// LS Electric XG5000 project: 121대대(4-11-23)
// PLC NewPLC
// module base 0 slot 0: 16점 예약 할당:XG-IN16
// module base 0 slot 1: Cnet:XGL-CH2A/B (Cnet 통신 모듈(RS-232C, RS-422/485))
// module base 0 slot 2: 아날로그입력 모듈:XGF-AC8A (A/D 전류 입력형 8채널)
// module base 0 slot 3: 입력 모듈:XGI-D24A/B (DC 24V 입력, 32점 (전류소스 싱크공용/ 전류소스 입력))
// module base 0 slot 4: 출력 모듈:XGQ-TR4A/B (트랜지스터 출력, 32점 (0.1A용, 싱크출력/소스출력))
// module base 0 slot 5: 고속카운터 모듈:XGF-HO2A (고속카운터 펄스(OC) 입력형, 2채널)

PROGRAM Sequence_Program (task: 스캔 프로그램)

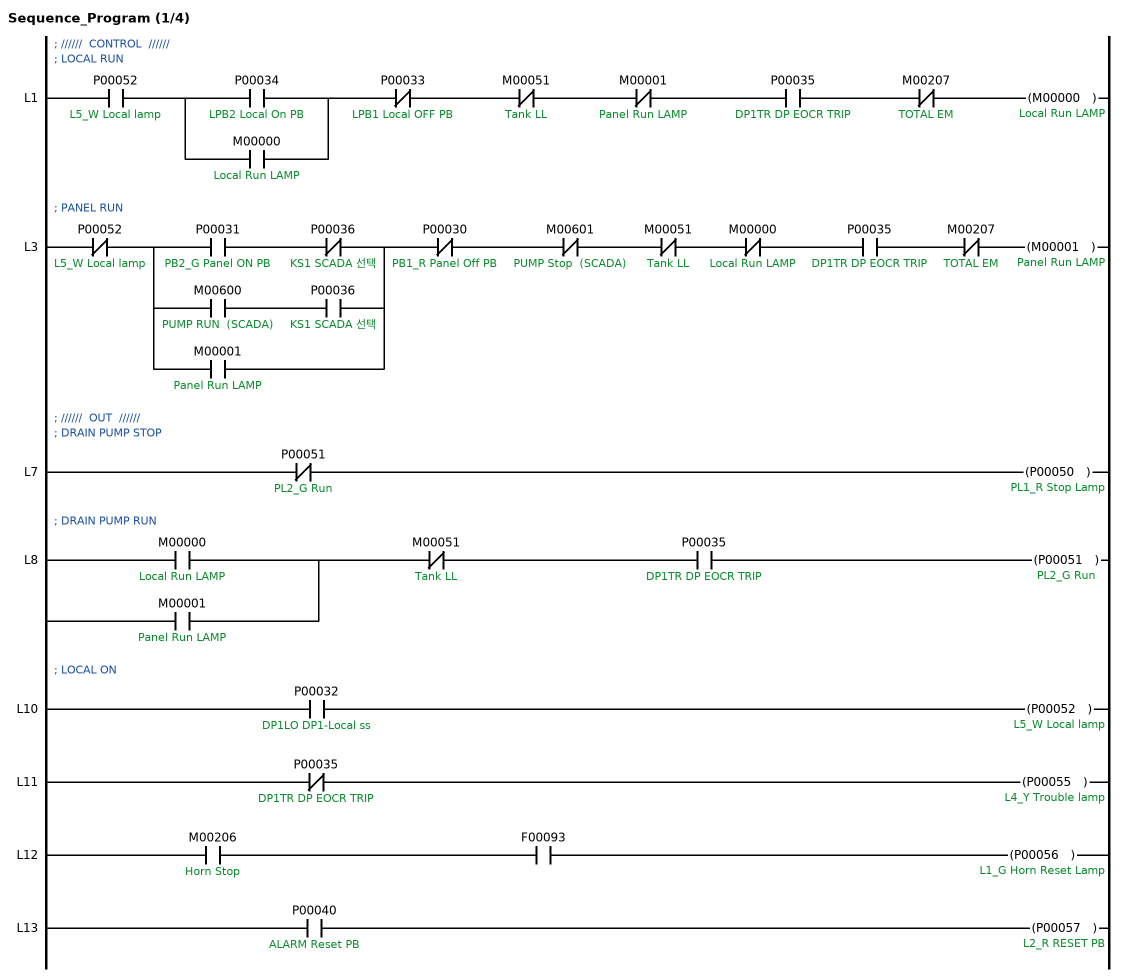
//      //////  CONTROL  //////
; L1
LOAD      P00052	// L5_W Local lamp
LOAD      P00034	// LPB2 Local On PB
OR        M00000	// Local Run LAMP
AND LOAD
AND NOT   P00033	// LPB1 Local OFF PB
AND NOT   M00051	// Tank LL
AND NOT   M00001	// Panel Run LAMP
AND       P00035	// DP1TR DP EOCR TRIP
AND NOT   M00207	// TOTAL EM
OUT       M00000	// Local Run LAMP
// output comment: LOCAL RUN
; L3
LOAD NOT  P00052	// L5_W Local lamp
LOAD      P00031	// PB2_G Panel ON PB
AND NOT   P00036	// KS1 SCADA 선택
LOAD      M00600	//   PUMP RUN  (SCADA)
AND       P00036	// KS1 SCADA 선택
OR LOAD
OR        M00001	// Panel Run LAMP
AND LOAD
AND NOT   P00030	// PB1_R Panel Off PB
AND NOT   M00601	//   PUMP Stop  (SCADA)
AND NOT   M00051	// Tank LL
AND NOT   M00000	// Local Run LAMP
AND       P00035	// DP1TR DP EOCR TRIP
AND NOT   M00207	// TOTAL EM
OUT       M00001	// Panel Run LAMP
// output comment: PANEL RUN
//      //////  OUT  //////
; L7
LOAD NOT  P00051	// PL2_G Run
OUT       P00050	// PL1_R Stop Lamp
// output comment: DRAIN PUMP STOP
; L8
LOAD      M00000	// Local Run LAMP
OR        M00001	// Panel Run LAMP
AND NOT   M00051	// Tank LL
AND       P00035	// DP1TR DP EOCR TRIP
OUT       P00051	// PL2_G Run
// output comment: DRAIN PUMP RUN
; L10
LOAD      P00032	// DP1LO DP1-Local ss
OUT       P00052	// L5_W Local lamp
// output comment: LOCAL ON
; L11
LOAD NOT  P00035	// DP1TR DP EOCR TRIP
OUT       P00055	// L4_Y Trouble lamp
// output comment: 
; L12
LOAD      M00206	// Horn Stop
AND       F00093
OUT       P00056	// L1_G Horn Reset Lamp
// output comment: 
; L13
LOAD      P00040	// ALARM Reset PB
OUT       P00057	// L2_R RESET PB
// output comment: 

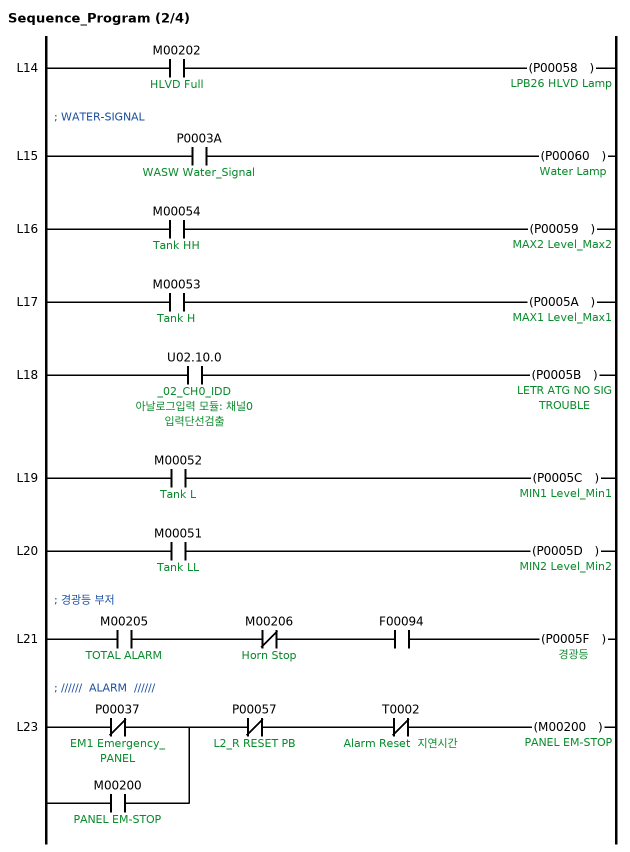
; L14
LOAD      M00202	// HLVD Full
OUT       P00058	// LPB26 HLVD Lamp
; L15
LOAD      P0003A	// WASW Water_Signal
OUT       P00060	// Water Lamp
// output comment: WATER-SIGNAL
; L16
LOAD      M00054	// Tank HH
OUT       P00059	// MAX2 Level_Max2
; L17
LOAD      M00053	// Tank H
OUT       P0005A	// MAX1 Level_Max1
; L18
LOAD      U02.10.0	// _02_CH0_IDD 아날로그입력 모듈: 채널0 입력단선검출
OUT       P0005B	// LETR ATG NO SIG TROUBLE
; L19
LOAD      M00052	// Tank L
OUT       P0005C	// MIN1 Level_Min1
; L20
LOAD      M00051	// Tank LL
OUT       P0005D	// MIN2 Level_Min2
; L21
LOAD      M00205	// TOTAL ALARM
AND NOT   M00206	// Horn Stop
AND       F00094
OUT       P0005F	// 경광등
// output comment: 경광등 부저
//      //////  ALARM  //////
; L23
LOAD NOT  P00037	// EM1 Emergency_PANEL
OR        M00200	// PANEL EM-STOP
AND NOT   P00057	// L2_R RESET PB
AND NOT   T0002	//   Alarm Reset  지연시간
OUT       M00200	// PANEL EM-STOP

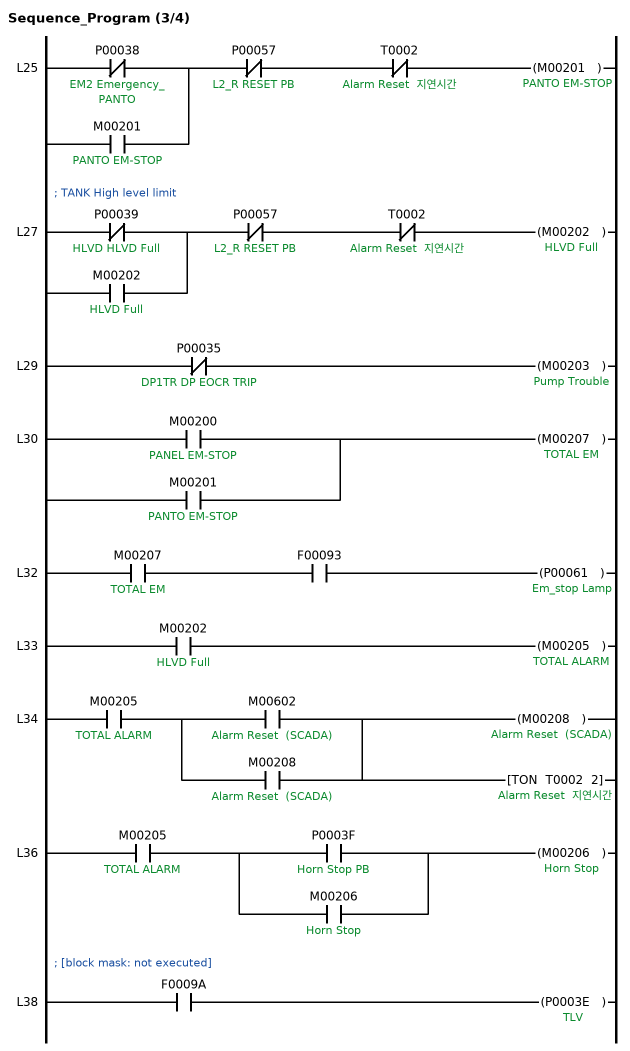
; L25
LOAD NOT  P00038	// EM2 Emergency_PANTO
OR        M00201	// PANTO EM-STOP
AND NOT   P00057	// L2_R RESET PB
AND NOT   T0002	//   Alarm Reset  지연시간
OUT       M00201	// PANTO EM-STOP
; L27
LOAD NOT  P00039	// HLVD HLVD Full
OR        M00202	// HLVD Full
AND NOT   P00057	// L2_R RESET PB
AND NOT   T0002	//   Alarm Reset  지연시간
OUT       M00202	// HLVD Full
// output comment: TANK High level limit
; L29
LOAD NOT  P00035	// DP1TR DP EOCR TRIP
OUT       M00203	// Pump Trouble
; L30
LOAD      M00200	// PANEL EM-STOP
OR        M00201	// PANTO EM-STOP
OUT       M00207	// TOTAL EM
; L32
LOAD      M00207	// TOTAL EM
AND       F00093
OUT       P00061	// Em_stop Lamp
; L33
LOAD      M00202	// HLVD Full
OUT       M00205	// TOTAL ALARM
; L34
LOAD      M00205	// TOTAL ALARM
LOAD      M00602	//   Alarm Reset  (SCADA)
OR        M00208	//   Alarm Reset  (SCADA)
AND LOAD
OUT       M00208	//   Alarm Reset  (SCADA)
TON       T0002 2	//   Alarm Reset  지연시간
; L36
LOAD      M00205	// TOTAL ALARM
LOAD      P0003F	// Horn Stop PB
OR        M00206	// Horn Stop
AND LOAD
OUT       M00206	// Horn Stop
; L38 (block mask: not executed)
LOAD      F0009A
OUT       P0003E	// TLV

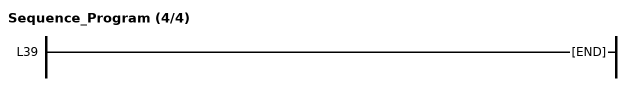
; L39
END

PROGRAM Analog (task: 스캔 프로그램)

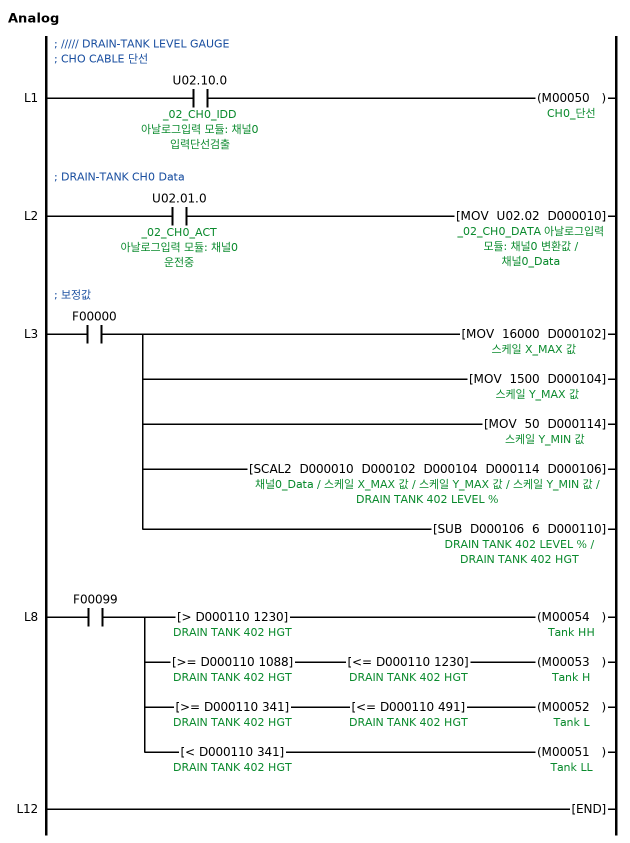
// ///// DRAIN-TANK LEVEL GAUGE
; L1
LOAD      U02.10.0	// _02_CH0_IDD 아날로그입력 모듈: 채널0 입력단선검출
OUT       M00050	// CH0_단선
// output comment: CHO CABLE 단선
; L2
LOAD      U02.01.0	// _02_CH0_ACT 아날로그입력 모듈: 채널0 운전중
MOV       U02.02 D000010	// _02_CH0_DATA 아날로그입력 모듈: 채널0 변환값 / 채널0_Data
// output comment: DRAIN-TANK CH0 Data
; L3
LOAD      F00000
MOV       16000 D000102	// 스케일 X_MAX 값
MOV       1500 D000104	// 스케일 Y_MAX 값
MOV       50 D000114	// 스케일 Y_MIN 값
SCAL2     D000010 D000102 D000104 D000114 D000106	// 채널0_Data / 스케일 X_MAX 값 / 스케일 Y_MAX 값 / 스케일 Y_MIN 값 / DRAIN TANK 402 LEVEL %
SUB       D000106 6 D000110	// DRAIN TANK 402 LEVEL % / DRAIN TANK 402 HGT
// output comment: 보정값
; L8
LOAD      F00099
MPUSH
AND>      D000110 1230	// DRAIN TANK 402 HGT
OUT       M00054	// Tank HH
MLOAD
AND>=     D000110 1088	// DRAIN TANK 402 HGT
AND<=     D000110 1230	// DRAIN TANK 402 HGT
OUT       M00053	// Tank H
MLOAD
AND>=     D000110 341	// DRAIN TANK 402 HGT
AND<=     D000110 491	// DRAIN TANK 402 HGT
OUT       M00052	// Tank L
MPOP
AND<      D000110 341	// DRAIN TANK 402 HGT
OUT       M00051	// Tank LL
; L12
END

PROGRAM Modbus-RTU_Comm (task: 스캔 프로그램)

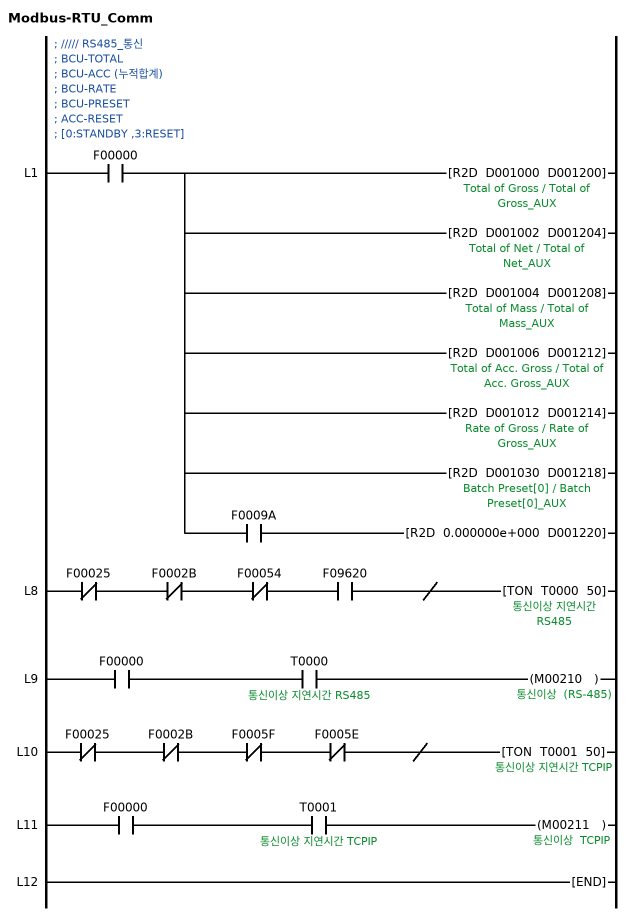
// ///// RS485_통신
; L1
LOAD      F00000
R2D       D001000 D001200	// Total of Gross / Total of Gross_AUX
R2D       D001002 D001204	// Total of Net / Total of Net_AUX
R2D       D001004 D001208	// Total of Mass / Total of Mass_AUX
R2D       D001006 D001212	// Total of Acc. Gross / Total of Acc. Gross_AUX
R2D       D001012 D001214	// Rate of Gross / Rate of Gross_AUX
R2D       D001030 D001218	// Batch Preset[0] / Batch Preset[0]_AUX
AND       F0009A
R2D       0.000000e+000 D001220
// output comment: BCU-TOTAL
// output comment: BCU-ACC (누적합계)
// output comment: BCU-RATE
// output comment: BCU-PRESET
// output comment: ACC-RESET [0:STANDBY ,3:RESET]
; L8
LOAD NOT  F00025
AND NOT   F0002B
AND NOT   F00054
AND       F09620
NOT
TON       T0000 50	// 통신이상 지연시간 RS485
; L9
LOAD      F00000
AND       T0000	// 통신이상 지연시간 RS485
OUT       M00210	// 통신이상  (RS-485)
; L10
LOAD NOT  F00025
AND NOT   F0002B
AND NOT   F0005F
AND NOT   F0005E
NOT
TON       T0001 50	// 통신이상 지연시간 TCPIP
; L11
LOAD      F00000
AND       T0001	// 통신이상 지연시간 TCPIP
OUT       M00211	// 통신이상  TCPIP
; L12
END

PROGRAM Flow_LIU (task: 스캔 프로그램)

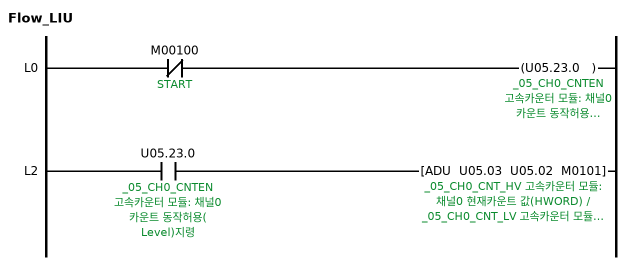
; L0
LOAD NOT  M00100	// START
OUT       U05.23.0	// _05_CH0_CNTEN 고속카운터 모듈: 채널0 카운트 동작허용(Level)지령
; L2
LOAD      U05.23.0	// _05_CH0_CNTEN 고속카운터 모듈: 채널0 카운트 동작허용(Level)지령
ADU       U05.03 U05.02 M0101	// _05_CH0_CNT_HV 고속카운터 모듈: 채널0 현재카운트 값(HWORD) / _05_CH0_CNT_LV 고속카운터 모듈: 채널0 현재카운트 값(LWORD)

VARIABLES AND COMMENTS (devices not used above)
P00053	BIT	LPL1 // DP1-Local Off lamp
P00054	BIT	LPL2 // DP1-Local Run lamp
P0005E	BIT	Em_stop
D00011	WORD	CH1_Data
M00055	BIT	Water
M01000	BIT	모드버스 블럭0 동작
M01010	BIT	모드버스 블럭 4동작
P0003B	BIT	PSW1
M00002	BIT	Valve_P1
P0003C	BIT	PSW2
M00003	BIT	Valve_P2
P0003D	BIT	GOCR
M00603	BIT	Horn Stop (SCADA)
M00209	BIT	TOTAL ALARM
D00108	WORD	DRAIN TANK 401 VOL
M00212	BIT	em test